{attribute addProperty BoxType "EL9576-0000-0016"}
{attribute addProperty Id "BCT_InputsAT %I*BCT_Inputs_BC823498120150WcStateAT %I*WcState_F855686C1620InfoDataAT %I*InfoData_BC63D37F80100"}
{attribute addProperty CRC "2162282512"}
{attribute addProperty SizeInBites "216"}
{attribute addProperty SizeInBytes "27"}
TYPE EL9576_4694F567 :
STRUCT
	{attribute addProperty Name "BCT_Inputs"}
	BCT_Inputs : BCT_Inputs_BC823498;
	{attribute addProperty Name "WcState"}
	WcState : WcState_F855686C;
	{attribute addProperty Name "InfoData"}
	InfoData : InfoData_BC63D37F;
END_STRUCT
END_TYPE

(* stored: Version 1.2.0.0, ProductVersion 3.1.4024.9
   DUT EL9576_4694F567: Id {68eab1fd-71aa-4038-b590-9800f7ef9cb5} *)
